TYPE STATE:
    STRUCT
        curTime: LREAL;
        dvar_M_p_x AT %Q*: DINT;
        cvar_M_p_t AT %Q*: LREAL;
    END_STRUCT
END_TYPE

(* stored: ProductVersion 3.1.0.18, Version 1.1.0.1 *)
